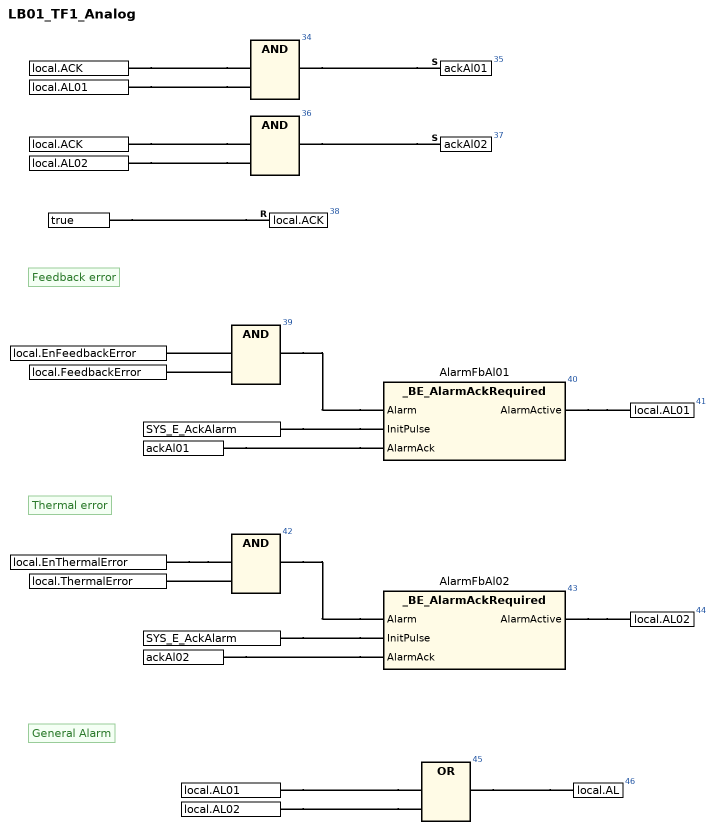
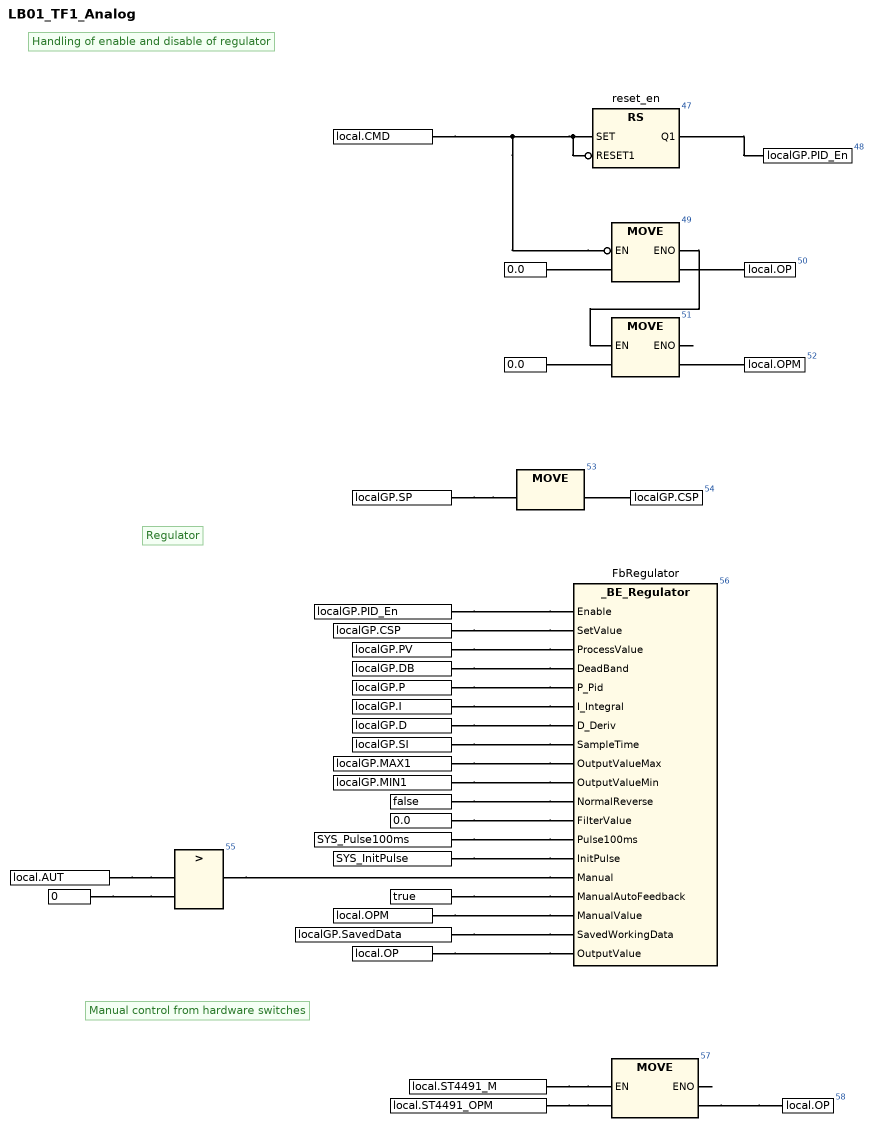
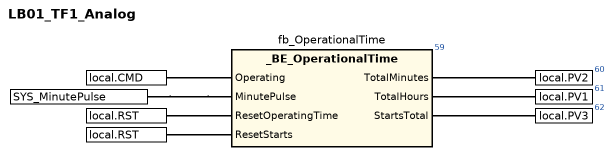
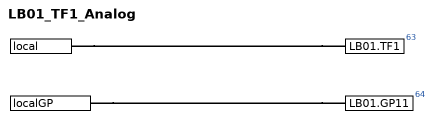
local := LB01.TF1;
localGP := LB01.GP11;
fanGuardOk := LB01.GP13.V;
local.EnFeedbackError := local.SP4 > 0;
local.EnThermalError := local.SP2 > 0;
local.EnFanGuardError := local.SP3 > 0;
_BE_Fan2(
    AutoStart := LB01.GeneralStart OR LB01.NH.V,
    AutoStartTimeDelay := local.SP1 + 5,
    BlockAutoStart := false,
    RunIndication := local.V,
    EnableFeedbackAlarm := local.EnFeedbackError,
    FeedbackAlarmTimeDelay := local.SP4,
    EnableThermicRelayAlarm := local.EnThermalError,
    ThermicRelayOk := local.ThermoRelay1,
    ThermicRelayAlarmTimeDelay := local.SP2,
    EnableFanGuardAlarm := local.EnFanGuardError,
    FanGuardOk := fanGuardOk,
    FanGuardAlarmTimeDelay := local.SP3,
    AlarmIndication := local.AL,
    AutoReg := local.AUT); // _BE_Fan_2
local.CMD := _BE_Fan2.StartSignalOutput;
local.FeedbackError := _BE_Fan2.FeedbackAlarm;
local.ThermalError := _BE_Fan2.ThermicRelayAlarm;
local.FanGuardError := _BE_Fan2.FanGuardAlarm;
// Manual control from hardware switches
local.Symbol := SEL(local.ST2792_M OR local.ST4491_M, SEL(_BE_Fan2.Status = 1 AND local.OP < 0.5, _BE_Fan2.Status, 0), SEL(local.ST2792_MCMD AND (local.ST4491_OPM > 0.5 AND local.ST4491_M), 0, 1));
local.Operating := local.CMD;
// HMI symbol for the handsymbol in iX
local.Symbol_M := 0;
IF local.AUT > 0 OR local.ST2792_M OR local.ST4491_M THEN _w1 := 1; END_IF
local.Symbol_M := _w1;
ackAl01 S= local.ACK AND local.AL01;
ackAl02 S= local.ACK AND local.AL02;
local.ACK R= true;
// Feedback error
AlarmFbAl01(
    Alarm := local.EnFeedbackError AND local.FeedbackError,
    InitPulse := SYS_E_AckAlarm,
    AlarmAck := ackAl01); // _BE_AlarmAckRequired
local.AL01 := AlarmFbAl01.AlarmActive;
// Thermal error
AlarmFbAl02(
    Alarm := local.EnThermalError AND local.ThermalError,
    InitPulse := SYS_E_AckAlarm,
    AlarmAck := ackAl02); // _BE_AlarmAckRequired
local.AL02 := AlarmFbAl02.AlarmActive;
// General Alarm
local.AL := local.AL01 OR local.AL02;
// Handling of enable and disable of regulator
reset_en(SET := local.CMD, RESET1 := NOT local.CMD); // RS
localGP.PID_En := reset_en.Q1;
_w2 := NOT local.CMD;
IF _w2 THEN _w3 := 0.0; END_IF
local.OP := _w3;
IF _w2 THEN _w4 := 0.0; END_IF
local.OPM := _w4;
localGP.CSP := localGP.SP;
// Regulator
FbRegulator(
    Enable := localGP.PID_En,
    SetValue := localGP.CSP,
    ProcessValue := localGP.PV,
    DeadBand := localGP.DB,
    P_Pid := localGP.P,
    I_Integral := localGP.I,
    D_Deriv := localGP.D,
    SampleTime := localGP.SI,
    OutputValueMax := localGP.MAX1,
    OutputValueMin := localGP.MIN1,
    NormalReverse := false,
    FilterValue := 0.0,
    Pulse100ms := SYS_Pulse100ms,
    InitPulse := SYS_InitPulse,
    Manual := local.AUT > 0,
    ManualAutoFeedback := true,
    ManualValue := local.OPM,
    SavedWorkingData := localGP.SavedData,
    OutputValue := local.OP); // _BE_Regulator
// Manual control from hardware switches
IF local.ST4491_M THEN _w5 := local.ST4491_OPM; END_IF
local.OP := _w5;
fb_OperationalTime(
    Operating := local.CMD,
    MinutePulse := SYS_MinutePulse,
    ResetOperatingTime := local.RST,
    ResetStarts := local.RST); // _BE_OperationalTime
local.PV2 := fb_OperationalTime.TotalMinutes;
local.PV1 := fb_OperationalTime.TotalHours;
local.PV3 := fb_OperationalTime.StartsTotal;
LB01.TF1 := local;
LB01.GP11 := localGP;

END_PROGRAM

// Device/AREA1/B001/LB01/Fan/FF1/LB01_FF1_Analog
PROGRAM LB01_FF1_Analog
VAR
	local:strFan_Analog;
	localGP:strSensor2_Regulator;
	ControlFan: _BE_Fan;
	FbRegulator: _BE_Regulator;
	_BE_Fan2: _BE_Fan_2;
	reset_en: RS;
	AlarmFbAl01: _BE_AlarmAckRequired;
	AlarmFbAl02: _BE_AlarmAckRequired;
	fb_OperationalTime: _BE_OperationalTime;
	ackAl01: BOOL;
	ackAl02: BOOL;
	fanGuardOk: BOOL;
END_VAR
VAR // added by the converter: edge detectors and wires of the graphical bodies
    _w1, _w3, _w4, _w5 : ANY;
    _w2 : BOOL;
END_VAR

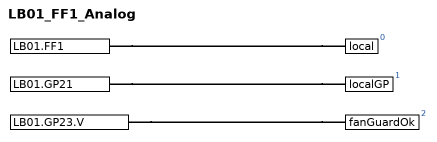
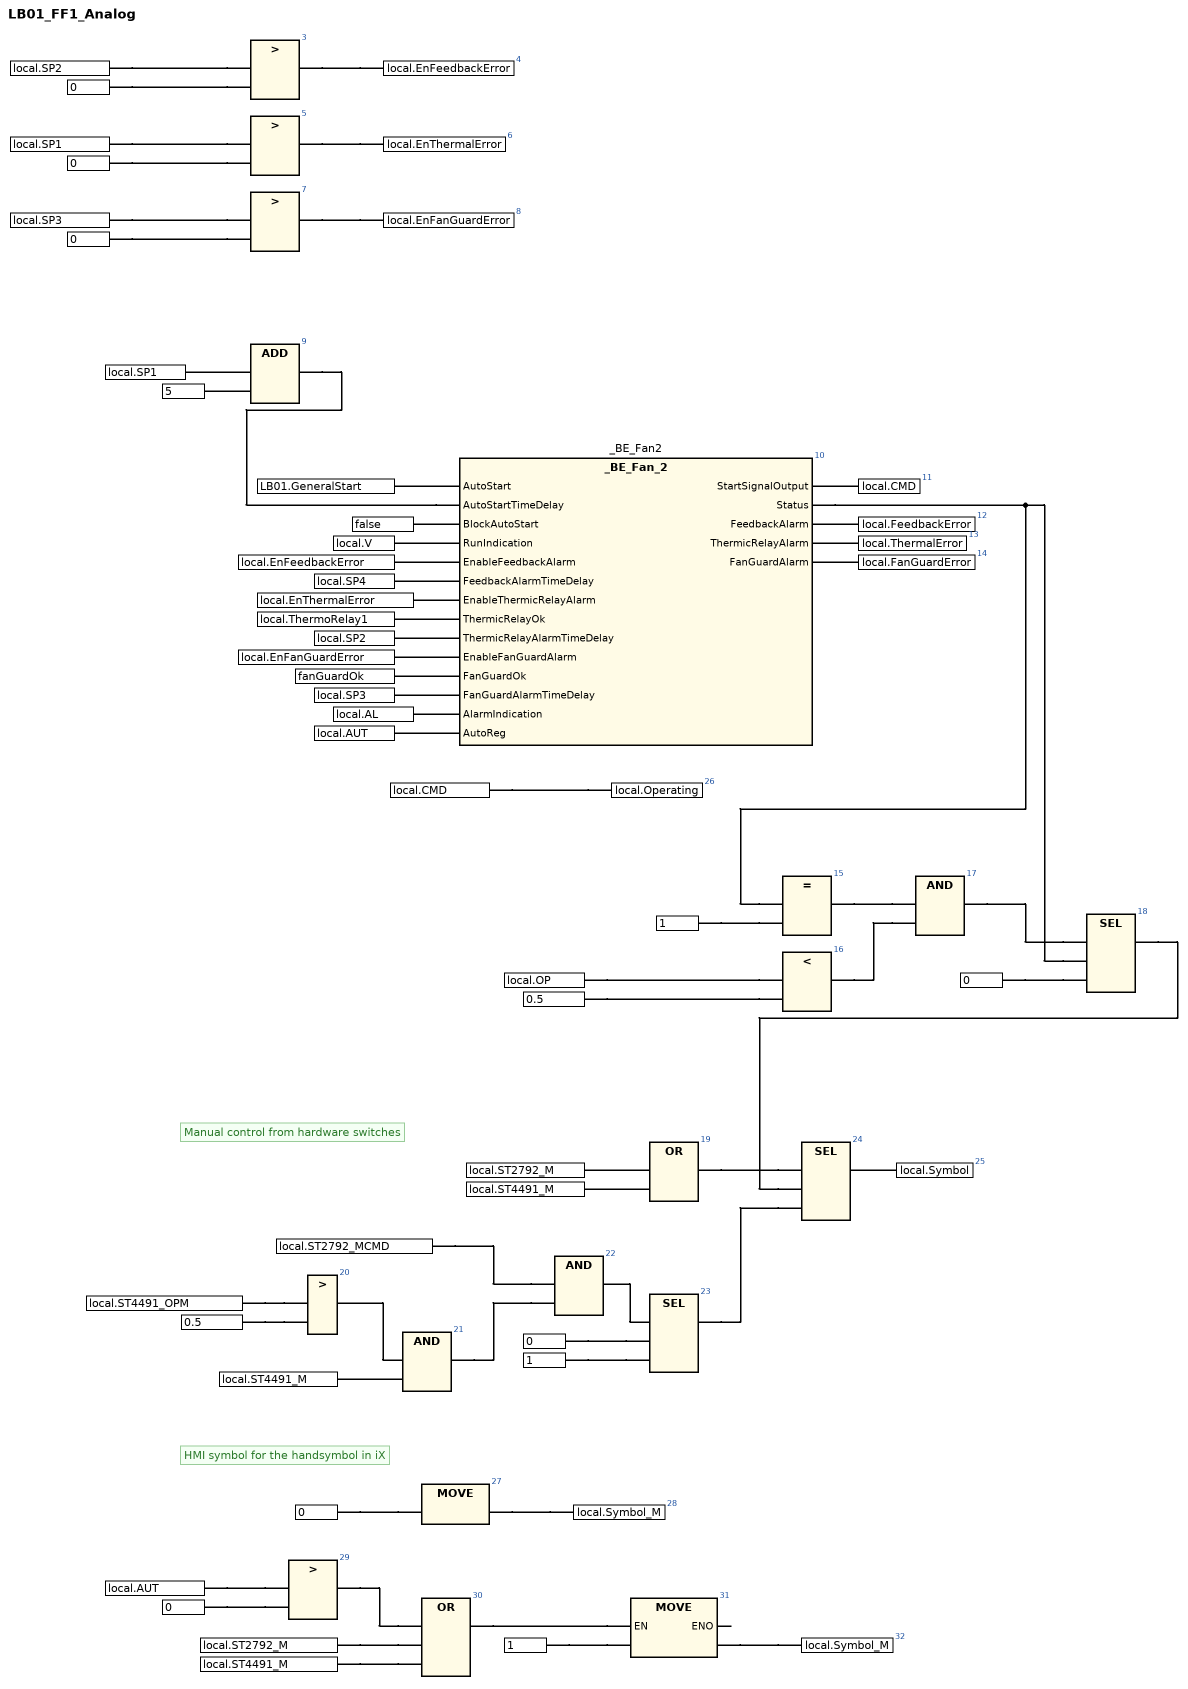
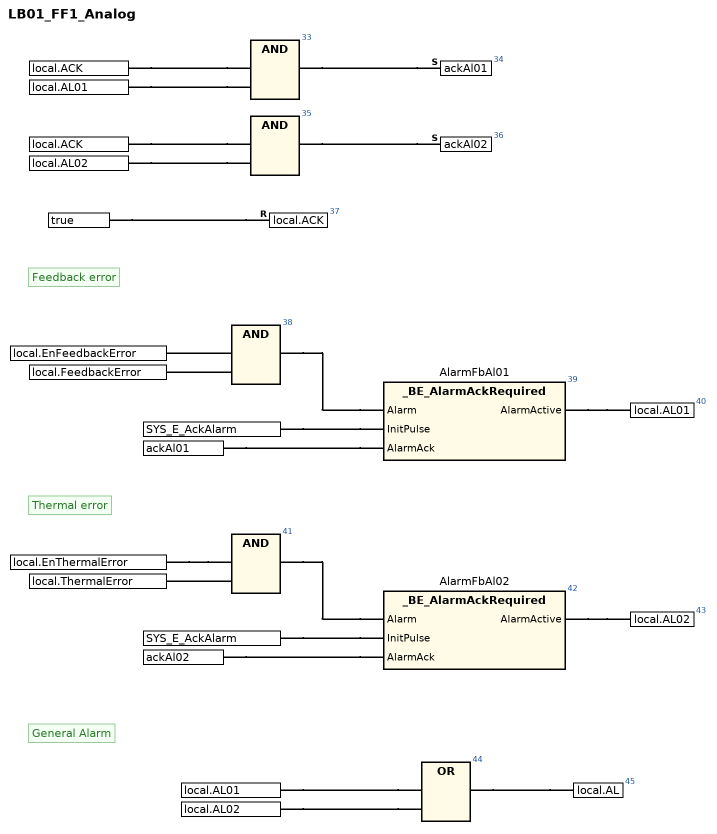
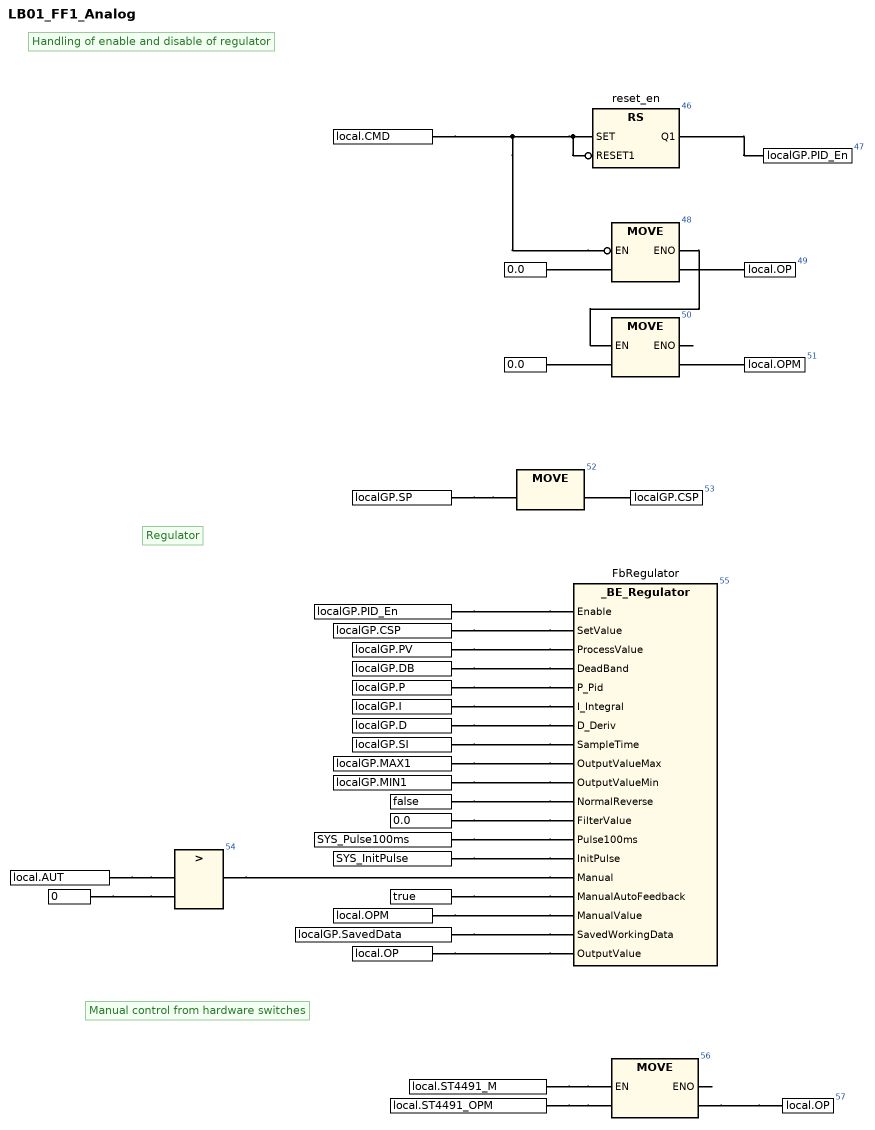
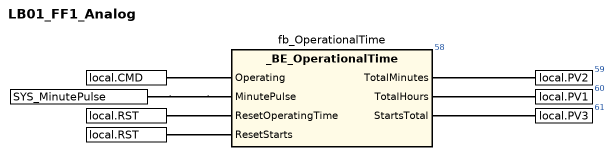
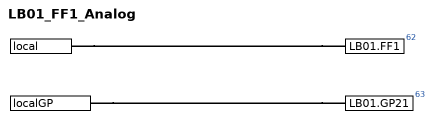
local := LB01.FF1;
localGP := LB01.GP21;
fanGuardOk := LB01.GP23.V;
local.EnFeedbackError := local.SP2 > 0;
local.EnThermalError := local.SP1 > 0;
local.EnFanGuardError := local.SP3 > 0;
_BE_Fan2(
    AutoStart := LB01.GeneralStart,
    AutoStartTimeDelay := local.SP1 + 5,
    BlockAutoStart := false,
    RunIndication := local.V,
    EnableFeedbackAlarm := local.EnFeedbackError,
    FeedbackAlarmTimeDelay := local.SP4,
    EnableThermicRelayAlarm := local.EnThermalError,
    ThermicRelayOk := local.ThermoRelay1,
    ThermicRelayAlarmTimeDelay := local.SP2,
    EnableFanGuardAlarm := local.EnFanGuardError,
    FanGuardOk := fanGuardOk,
    FanGuardAlarmTimeDelay := local.SP3,
    AlarmIndication := local.AL,
    AutoReg := local.AUT); // _BE_Fan_2
local.CMD := _BE_Fan2.StartSignalOutput;
local.FeedbackError := _BE_Fan2.FeedbackAlarm;
local.ThermalError := _BE_Fan2.ThermicRelayAlarm;
local.FanGuardError := _BE_Fan2.FanGuardAlarm;
// Manual control from hardware switches
local.Symbol := SEL(local.ST2792_M OR local.ST4491_M, SEL(_BE_Fan2.Status = 1 AND local.OP < 0.5, _BE_Fan2.Status, 0), SEL(local.ST2792_MCMD AND (local.ST4491_OPM > 0.5 AND local.ST4491_M), 0, 1));
local.Operating := local.CMD;
// HMI symbol for the handsymbol in iX
local.Symbol_M := 0;
IF local.AUT > 0 OR local.ST2792_M OR local.ST4491_M THEN _w1 := 1; END_IF
local.Symbol_M := _w1;
ackAl01 S= local.ACK AND local.AL01;
ackAl02 S= local.ACK AND local.AL02;
local.ACK R= true;
// Feedback error
AlarmFbAl01(
    Alarm := local.EnFeedbackError AND local.FeedbackError,
    InitPulse := SYS_E_AckAlarm,
    AlarmAck := ackAl01); // _BE_AlarmAckRequired
local.AL01 := AlarmFbAl01.AlarmActive;
// Thermal error
AlarmFbAl02(
    Alarm := local.EnThermalError AND local.ThermalError,
    InitPulse := SYS_E_AckAlarm,
    AlarmAck := ackAl02); // _BE_AlarmAckRequired
local.AL02 := AlarmFbAl02.AlarmActive;
// General Alarm
local.AL := local.AL01 OR local.AL02;
// Handling of enable and disable of regulator
reset_en(SET := local.CMD, RESET1 := NOT local.CMD); // RS
localGP.PID_En := reset_en.Q1;
_w2 := NOT local.CMD;
IF _w2 THEN _w3 := 0.0; END_IF
local.OP := _w3;
IF _w2 THEN _w4 := 0.0; END_IF
local.OPM := _w4;
localGP.CSP := localGP.SP;
// Regulator
FbRegulator(
    Enable := localGP.PID_En,
    SetValue := localGP.CSP,
    ProcessValue := localGP.PV,
    DeadBand := localGP.DB,
    P_Pid := localGP.P,
    I_Integral := localGP.I,
    D_Deriv := localGP.D,
    SampleTime := localGP.SI,
    OutputValueMax := localGP.MAX1,
    OutputValueMin := localGP.MIN1,
    NormalReverse := false,
    FilterValue := 0.0,
    Pulse100ms := SYS_Pulse100ms,
    InitPulse := SYS_InitPulse,
    Manual := local.AUT > 0,
    ManualAutoFeedback := true,
    ManualValue := local.OPM,
    SavedWorkingData := localGP.SavedData,
    OutputValue := local.OP); // _BE_Regulator
// Manual control from hardware switches
IF local.ST4491_M THEN _w5 := local.ST4491_OPM; END_IF
local.OP := _w5;
fb_OperationalTime(
    Operating := local.CMD,
    MinutePulse := SYS_MinutePulse,
    ResetOperatingTime := local.RST,
    ResetStarts := local.RST); // _BE_OperationalTime
local.PV2 := fb_OperationalTime.TotalMinutes;
local.PV1 := fb_OperationalTime.TotalHours;
local.PV3 := fb_OperationalTime.StartsTotal;
LB01.FF1 := local;
LB01.GP21 := localGP;

END_PROGRAM

// Device/AREA1/B001/LB01/Pump/P2/LB01_P2
PROGRAM LB01_P2
VAR
	local:strPumpExercise;
	fbControlPump2: _BE_Pump_2;
	fbPumpStartCondition: _BE_PumpStartConditions;
	fb_OperationalTime: _BE_OperationalTime;
	fbExercise: _BE_Exercise;
	ackAl01: BOOL;
	ackAl02: BOOL;
	sv_op: REAL;
	startPump: BOOL;
	AlarmFbAL01: _BE_AlarmAckRequired;
	AlarmFbAL02: _BE_AlarmAckRequired;
END_VAR
VAR // added by the converter: edge detectors and wires of the graphical bodies
    _w1 : ANY;
END_VAR

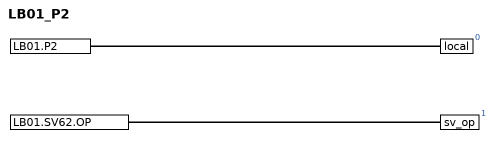
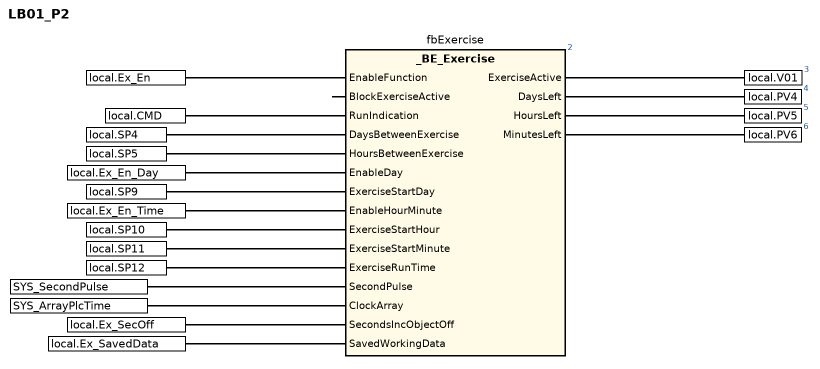
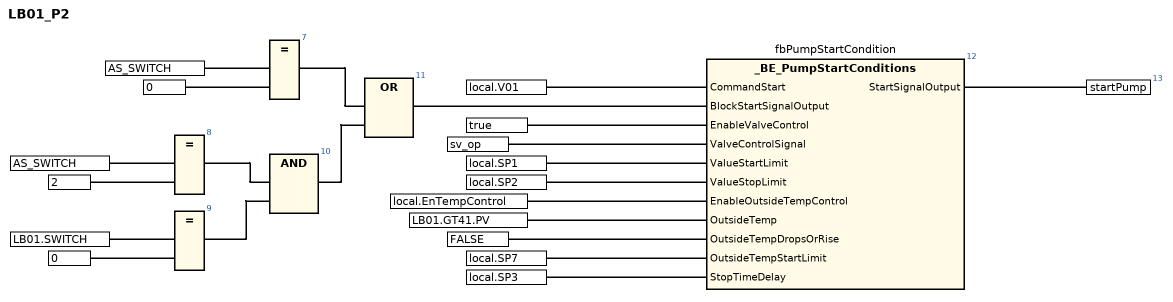
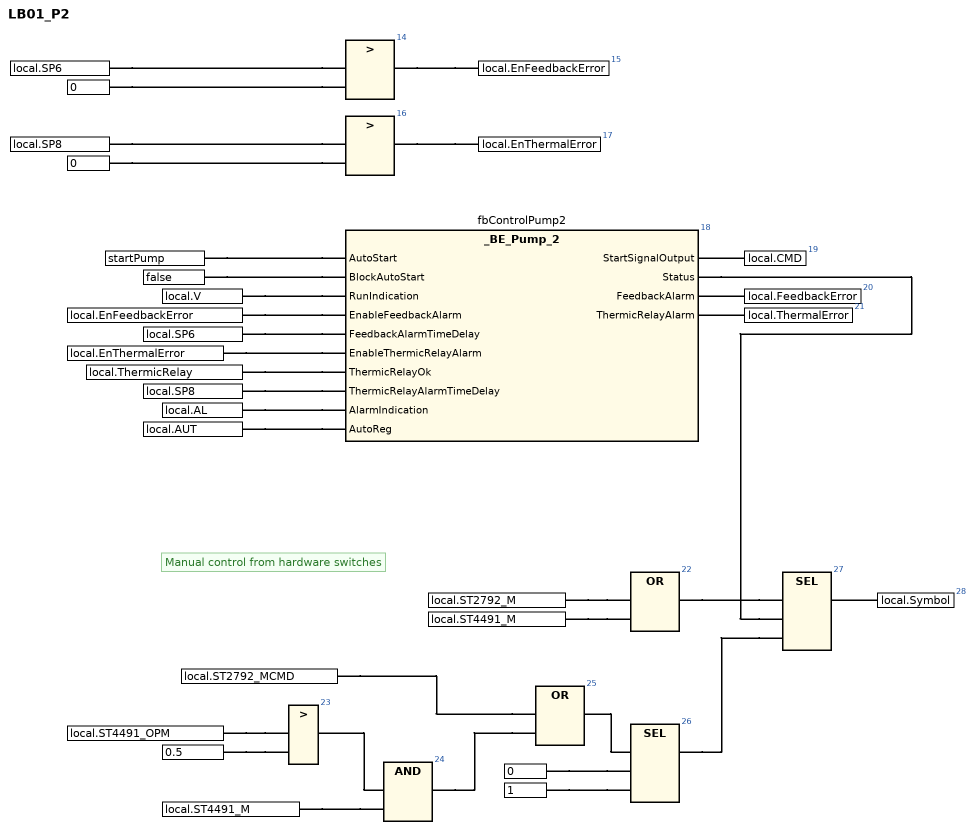
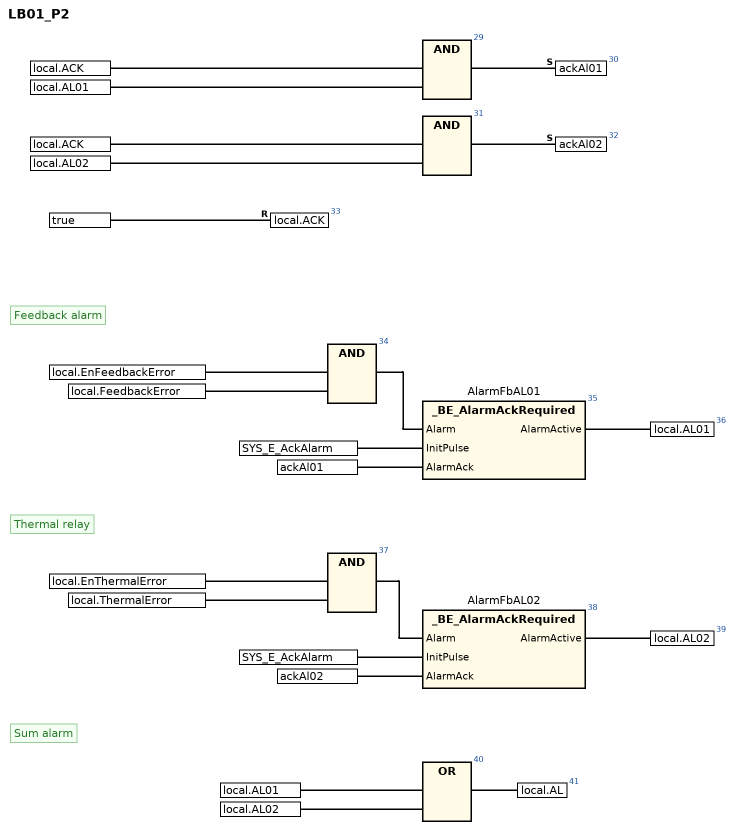
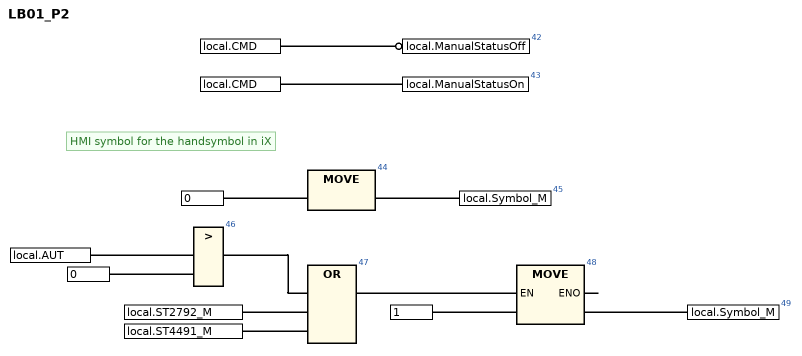
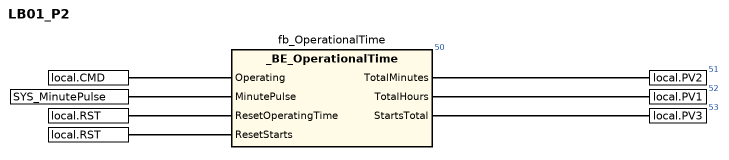
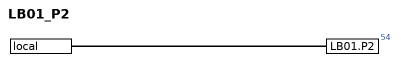
local := LB01.P2;
sv_op := LB01.SV62.OP;
fbExercise(
    EnableFunction := local.Ex_En,
    RunIndication := local.CMD,
    DaysBetweenExercise := local.SP4,
    HoursBetweenExercise := local.SP5,
    EnableDay := local.Ex_En_Day,
    ExerciseStartDay := local.SP9,
    EnableHourMinute := local.Ex_En_Time,
    ExerciseStartHour := local.SP10,
    ExerciseStartMinute := local.SP11,
    ExerciseRunTime := local.SP12,
    SecondPulse := SYS_SecondPulse,
    ClockArray := SYS_ArrayPlcTime,
    SecondsIncObjectOff := local.Ex_SecOff,
    SavedWorkingData := local.Ex_SavedData); // _BE_Exercise
local.V01 := fbExercise.ExerciseActive;
local.PV4 := fbExercise.DaysLeft;
local.PV5 := fbExercise.HoursLeft;
local.PV6 := fbExercise.MinutesLeft;
fbPumpStartCondition(
    CommandStart := local.V01,
    BlockStartSignalOutput := AS_SWITCH = 0 OR AS_SWITCH = 2 AND LB01.SWITCH = 0,
    EnableValveControl := true,
    ValveControlSignal := sv_op,
    ValueStartLimit := local.SP1,
    ValueStopLimit := local.SP2,
    EnableOutsideTempControl := local.EnTempControl,
    OutsideTemp := LB01.GT41.PV,
    OutsideTempDropsOrRise := FALSE,
    OutsideTempStartLimit := local.SP7,
    StopTimeDelay := local.SP3); // _BE_PumpStartConditions
startPump := fbPumpStartCondition.StartSignalOutput;
local.EnFeedbackError := local.SP6 > 0;
local.EnThermalError := local.SP8 > 0;
fbControlPump2(
    AutoStart := startPump,
    BlockAutoStart := false,
    RunIndication := local.V,
    EnableFeedbackAlarm := local.EnFeedbackError,
    FeedbackAlarmTimeDelay := local.SP6,
    EnableThermicRelayAlarm := local.EnThermalError,
    ThermicRelayOk := local.ThermicRelay,
    ThermicRelayAlarmTimeDelay := local.SP8,
    AlarmIndication := local.AL,
    AutoReg := local.AUT); // _BE_Pump_2
local.CMD := fbControlPump2.StartSignalOutput;
local.FeedbackError := fbControlPump2.FeedbackAlarm;
local.ThermalError := fbControlPump2.ThermicRelayAlarm;
// Manual control from hardware switches
local.Symbol := SEL(local.ST2792_M OR local.ST4491_M, fbControlPump2.Status, SEL(local.ST2792_MCMD OR local.ST4491_OPM > 0.5 AND local.ST4491_M, 0, 1));
ackAl01 S= local.ACK AND local.AL01;
ackAl02 S= local.ACK AND local.AL02;
local.ACK R= true;
// Feedback alarm
AlarmFbAL01(
    Alarm := local.EnFeedbackError AND local.FeedbackError,
    InitPulse := SYS_E_AckAlarm,
    AlarmAck := ackAl01); // _BE_AlarmAckRequired
local.AL01 := AlarmFbAL01.AlarmActive;
// Thermal relay
AlarmFbAL02(
    Alarm := local.EnThermalError AND local.ThermalError,
    InitPulse := SYS_E_AckAlarm,
    AlarmAck := ackAl02); // _BE_AlarmAckRequired
local.AL02 := AlarmFbAL02.AlarmActive;
// Sum alarm
local.AL := local.AL01 OR local.AL02;
local.ManualStatusOff := NOT local.CMD;
local.ManualStatusOn := local.CMD;
// HMI symbol for the handsymbol in iX
local.Symbol_M := 0;
IF local.AUT > 0 OR local.ST2792_M OR local.ST4491_M THEN _w1 := 1; END_IF
local.Symbol_M := _w1;
fb_OperationalTime(
    Operating := local.CMD,
    MinutePulse := SYS_MinutePulse,
    ResetOperatingTime := local.RST,
    ResetStarts := local.RST); // _BE_OperationalTime
local.PV2 := fb_OperationalTime.TotalMinutes;
local.PV1 := fb_OperationalTime.TotalHours;
local.PV3 := fb_OperationalTime.StartsTotal;
LB01.P2 := local;

END_PROGRAM

// Device/AREA1/B001/LB01/Sensor/Pressure/GP11/LB01_GP11
PROGRAM LB01_GP11
VAR
	local:strSensor2_Regulator;
	gt_Min: TON;
	gt_Max: TON;
	reset_en: RS;
	ackLal: BOOL;
	ackHal: BOOL;
	AlarmAcknowledge01: _BE_AlarmAckRemote;
	AlarmAcknowledge02: _BE_AlarmAckRemote;
END_VAR
VAR // added by the converter: edge detectors and wires of the graphical bodies
    _w1, _w3 : ANY;
    _w2 : BOOL;
END_VAR

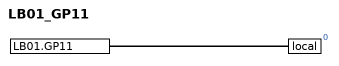
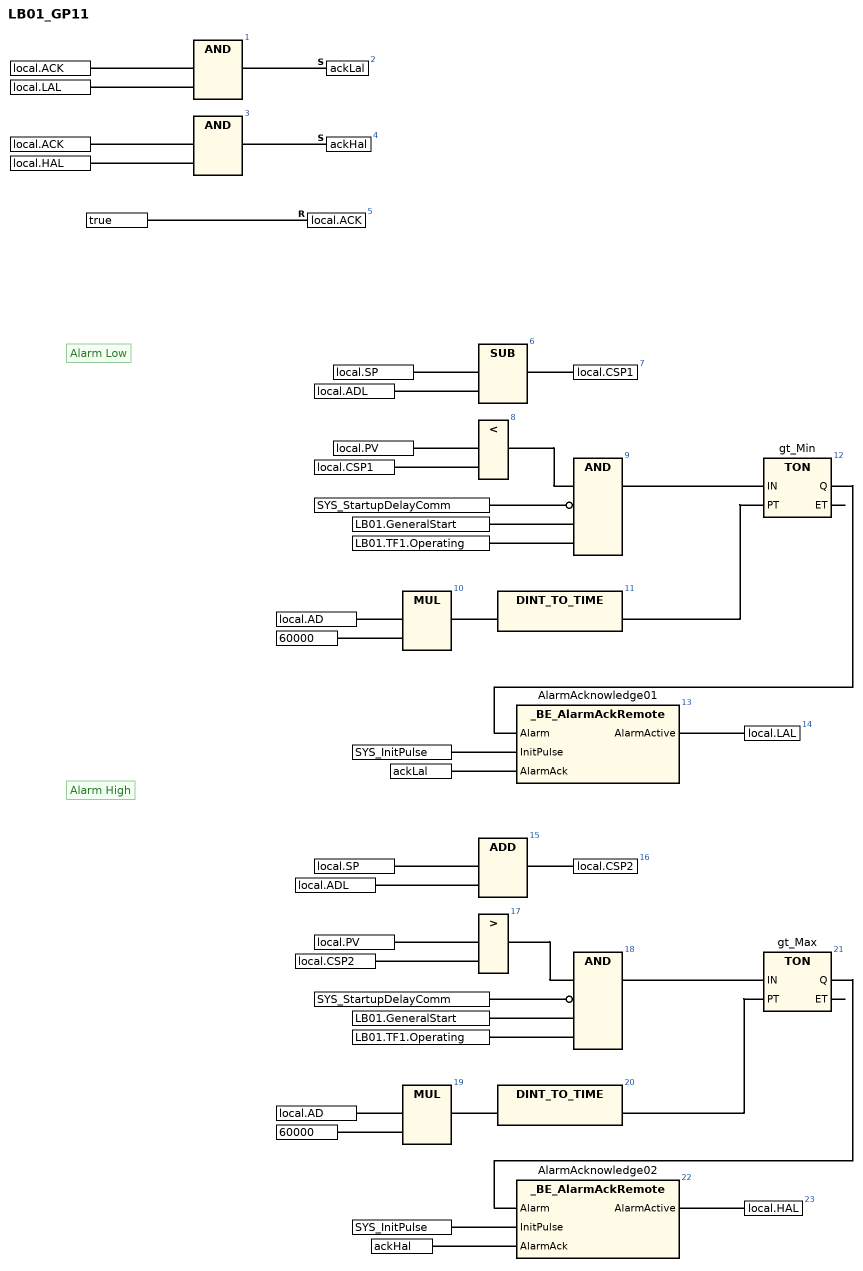
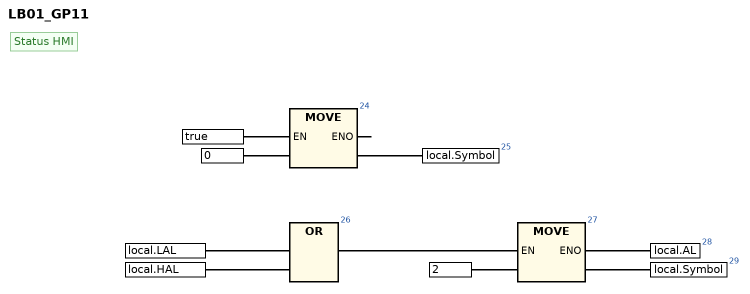
